FUNCTION_BLOCK FB_oscillatore
VAR_INPUT
	enable	: BOOL;
	t_high	: TIME;
	t_low	: TIME;	
END_VAR
VAR_OUTPUT
	q		: BOOL;	
END_VAR
VAR
	t1		: TON();
	t2		: TON();	
END_VAR

t1(in := enable AND NOT t2.Q, pt := t_low);
t2(in := t1.Q, pt := t_high);
// comando dell'uscita dell'oscillatore
q := t1.Q;

END_FUNCTION_BLOCK

(* stored: Version 1.1.0.1, ProductVersion 3.1.4024.12
   POU FB_oscillatore: Id {04152e5d-4d97-4702-ab11-291beaf6f3ff}, SpecialFunc None *)
